FUNCTION_BLOCK FuseChannelExtended EXTENDS FuseChannelBasic IMPLEMENTS IFuseChannelExtended
VAR_INPUT
END_VAR
VAR_OUTPUT
END_VAR
VAR
	_ChnEx : EL922x_ChannelExtended;
END_VAR


PROPERTY DisabledByDI : BOOL
GET
DisabledByDI := _ChnEx.Status.DisabledByDI;
END_GET
END_PROPERTY


PROPERTY DisabledByOutput : BOOL
GET
DisabledByOutput := _ChnEx.Status.DisabledByOutput;
END_GET
END_PROPERTY


PROPERTY DisabledBySwitch : BOOL
GET
DisabledBySwitch := _ChnEx.Status.DisabledBySwitch;
END_GET
END_PROPERTY


PROPERTY Overload : BOOL
GET
Overload := _ChnEx.Status.Overload;
END_GET
END_PROPERTY


PROPERTY Overvoltage : BOOL
GET
Overvoltage := _ChnEx.Status.Overvoltage;
END_GET
END_PROPERTY

{warning 'add property implementation'}
PROPERTY ShortCircuit : BOOL
GET
ShortCircuit := _ChnEx.Status.ShortCircuit;
END_GET
END_PROPERTY

{warning 'add property implementation'}
PROPERTY StateDeviceSwitch : BOOL
GET
StateDeviceSwitch := _ChnEx.Status.StateDeviceSwitch;
END_GET
END_PROPERTY

{warning 'add property implementation'}
PROPERTY StateDigitalInput : BOOL
GET
StateDigitalInput := _ChnEx.Status.StateDigitalInput;
END_GET
END_PROPERTY

{warning 'add property implementation'}
PROPERTY Undervoltage : BOOL
GET
Undervoltage := _ChnEx.Status.Undervoltage;
END_GET
END_PROPERTY

END_FUNCTION_BLOCK

(* stored: Version 1.1.0.1, ProductVersion 3.1.4024.6
   POU FuseChannelExtended: Id {4337dc67-16d6-41c8-a93d-58f4c5b5f6c3}, SpecialFunc None
   Property DisabledByDI: Id {aaa5413d-cae1-43bb-826f-64cdc481af58}
   Get Get: Id {46a43373-4ed2-49bd-9b0d-da57bae95df0}
   Property DisabledByOutput: Id {5d3de88f-7ec4-4ae0-8afd-ae81c12e5f09}
   Get Get: Id {21798a35-a777-4236-9d96-b20bc10f7fc9}
   Property DisabledBySwitch: Id {3bad2763-8f31-405d-a672-4e32aa8e76e6}
   Get Get: Id {8c65b039-5ce7-41ec-beb5-957afa167ca2}
   Property Overload: Id {0a399695-d904-44da-8a8c-d40025f0bae2}
   Get Get: Id {a48f0bd8-5b8d-40ca-9066-e8fa5988f50d}
   Property Overvoltage: Id {82f8afce-d30b-477d-9e0f-b28cc0598392}
   Get Get: Id {558dc962-f54c-4d89-be6f-913248366ab3}
   Property ShortCircuit: Id {e00036ed-5cf2-4d7d-9dbf-a2e92dcaa27a}
   Get Get: Id {a2926c79-64a7-4da1-b7a0-1139822534b3}
   Property StateDeviceSwitch: Id {62b2d540-cbd9-446e-8476-f480b4ddcec0}
   Get Get: Id {6a9fb8a3-db95-4b08-84f0-8e4671cf40ba}
   Property StateDigitalInput: Id {2a838b84-ca7e-4183-9966-b5a34ce0dd5b}
   Get Get: Id {3f8f32b1-238c-4aea-828e-6d26948742ae}
   Property Undervoltage: Id {bde0c85b-2023-4486-821c-9f50ba7bcff8}
   Get Get: Id {d45a69dc-1bef-4ddb-9b42-52e2b3f3ecc3} *)
